PROGRAM Visu_handling
VAR
END_VAR

(*IF GVL.visuOUT0 THEN
	GVL.X1_00 := TRUE;
ELSIF NOT GVL.visuOUT0 THEN
	GVL.X1_00 := FALSE;
END_IF
IF GVL.visuOUT1 THEN
	GVL.X1_01 := TRUE;
ELSIF NOT GVL.visuOUT1 THEN
	GVL.X1_01 := FALSE;
END_IF
IF GVL.visuOUT2 THEN
	GVL.X1_02 := TRUE;
ELSIF NOT GVL.visuOUT2 THEN
	GVL.X1_02 := FALSE;
END_IF
IF GVL.visuOUT3 THEN
	GVL.X1_03 := TRUE;
ELSIF NOT GVL.visuOUT3 THEN
	GVL.X1_03 := FALSE;
END_IF
IF GVL.visuOUT4 THEN
	GVL.X1_04 := TRUE;
ELSIF NOT GVL.visuOUT4 THEN
	GVL.X1_04 := FALSE;
END_IF
IF GVL.visuOUT5 THEN
	GVL.X1_05 := TRUE;
ELSIF NOT GVL.visuOUT5 THEN
	GVL.X1_05 := FALSE;
END_IF
IF GVL.visuOUT6 THEN
	GVL.X1_06 := TRUE;
ELSIF NOT GVL.visuOUT6 THEN
	GVL.X1_06 := FALSE;
END_IF
IF GVL.visuOUT7 THEN
	GVL.X1_07 := TRUE;
ELSIF NOT GVL.visuOUT7 THEN
	GVL.X1_07 := FALSE;
END_IF


IF GVL.visuOUT20 THEN
	GVL.X2_00 := TRUE;
ELSIF NOT GVL.visuOUT20 THEN
	GVL.X2_00 := FALSE;
END_IF
IF GVL.visuOUT21 THEN
	GVL.X2_01 := TRUE;
ELSIF NOT GVL.visuOUT21 THEN
	GVL.X2_01 := FALSE;
END_IF
IF GVL.visuOUT22 THEN
	GVL.X2_02 := TRUE;
ELSIF NOT GVL.visuOUT22 THEN
	GVL.X2_02 := FALSE;
END_IF
IF GVL.visuOUT23 THEN
	GVL.X2_03 := TRUE;
ELSIF NOT GVL.visuOUT23 THEN
	GVL.X2_03 := FALSE;
END_IF*)

END_PROGRAM

(* stored: Version 1.1.0.1, ProductVersion 3.1.4024.15
   POU Visu_handling: Id {bbf4b788-9069-45ef-b8b8-929ad6965378}, SpecialFunc None *)
